TYPE T_Position : DINT; END_TYPE

(* stored: Version 1.1.0.1
   DUT T_Position: Id {6eb3ac3e-30e1-094d-0b8e-c13e8e2957bb} *)
